// TIA Portal V17 export
// export: Created 2024-06-14T09:52:46.5071522Z, ExportSetting WithDefaults, DisplayName Totally Integrated Automation Portal, DisplayVersion V17, DisplayName TIA Portal Openness, DisplayVersion V17, DisplayName TIA Portal Version Control Interface, DisplayVersion V17, DisplayName Simotion SCOUT TIA, DisplayVersion 5.4.3.0, DisplayName SINAMICS Startdrive Advanced, DisplayVersion V17 SP1 Update 1, DisplayName SINAMICS Startdrive G110M, G120, G120C, G120D, G120P, G115D, DisplayVersion V17 SP1 Update 1, DisplayName SINAMICS Startdrive G130, G150, S120, S150, SINAMICS MV, S210, DisplayVersion V17 SP1 Update 1, DisplayName STEP 7 Professional, DisplayVersion V17, DisplayName STEP 7 Safety, DisplayVersion V17, DisplayName WinCC Professional, DisplayVersion V17
FUNCTION_BLOCK "Disable"   // FB3, LAD
{ S7_Optimized_Access := 'TRUE' }
VERSION : 0.1
// stored: AutoNumber false, IsIECCheckEnabled false, IsRetainMemResEnabled false, MemoryReserve 100, SetENOAutomatically false, UDAEnableTagReadback false
   VAR_INPUT
      Enable_Cylinder { ExternalAccessible := 'False'; ExternalVisible := 'False'; ExternalWritable := 'False'} : Array[1..6] of Bool;
      Enabled_Cylinder { ExternalAccessible := 'False'; ExternalVisible := 'False'; ExternalWritable := 'False'} : Int;
   END_VAR
   VAR_OUTPUT
      "First_Cylinder[1]" : Int;
      "First_Cylinder[2]" : Int;
      "First_Cylinder[3]" : Int;
      "First_Cylinder[4]" : Int;
      "First_Cylinder[5]" : Int;
      "First_Cylinder[6]" : Int;
      Disab_Total_Cyl : Int;
   END_VAR
   VAR
      Add_Cylinder : Array[1..6] of Int;
   END_VAR
   VAR_TEMP
      Temp8 : Int;
      Temp7 : Int;
      Temp6 : Int;
      Temp5 : Int;
      Temp4 : Int;
      Temp3 : Int;
      Temp2 : Int;
      Temp1 : Int;
      Temp9 : Int;
      Temp_8 : Int;
      Temp_7 : Int;
      Temp_6 : Int;
      Temp_5 : Int;
      Temp_4 : Int;
      Temp_3 : Int;
      Temp_2 : Int;
      Temp_1 : Int;
      Temp_9 : Int;
      Temp_91 : Int;
      Temp_81 : Int;
      Temp_71 : Int;
      Temp_61 : Int;
      Temp_51 : Int;
      Temp_41 : Int;
      Temp_31 : Int;
      Temp_21 : Int;
      Temp_11 : Int;
      Temp10 : Int;
      Temp_10 : Int;
      Temp_101 : Int;
   END_VAR
BEGIN

REGION Network 1: Disable Cylinder
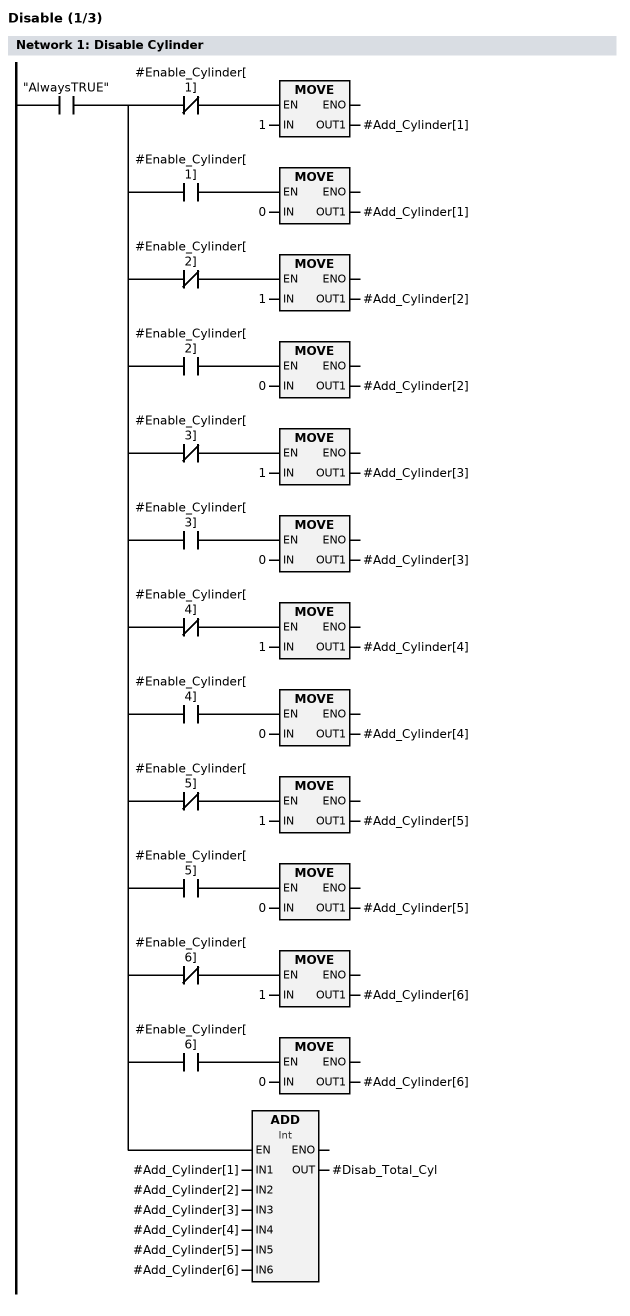
   RUNG wire#powerrail
      Contact( "AlwaysTRUE" )
      wire#w1
      I_Contact( #Enable_Cylinder[1] )
      Move(in := 1, out1 => #Add_Cylinder[1])
   END_RUNG
   RUNG wire#w1
      Contact( #Enable_Cylinder[1] )
      Move(in := 0, out1 => #Add_Cylinder[1])
   END_RUNG
   RUNG wire#w1
      I_Contact( #Enable_Cylinder[2] )
      Move(in := 1, out1 => #Add_Cylinder[2])
   END_RUNG
   RUNG wire#w1
      Contact( #Enable_Cylinder[2] )
      Move(in := 0, out1 => #Add_Cylinder[2])
   END_RUNG
   RUNG wire#w1
      I_Contact( #Enable_Cylinder[3] )
      Move(in := 1, out1 => #Add_Cylinder[3])
   END_RUNG
   RUNG wire#w1
      Contact( #Enable_Cylinder[3] )
      Move(in := 0, out1 => #Add_Cylinder[3])
   END_RUNG
   RUNG wire#w1
      I_Contact( #Enable_Cylinder[4] )
      Move(in := 1, out1 => #Add_Cylinder[4])
   END_RUNG
   RUNG wire#w1
      Contact( #Enable_Cylinder[4] )
      Move(in := 0, out1 => #Add_Cylinder[4])
   END_RUNG
   RUNG wire#w1
      I_Contact( #Enable_Cylinder[5] )
      Move(in := 1, out1 => #Add_Cylinder[5])
   END_RUNG
   RUNG wire#w1
      Contact( #Enable_Cylinder[5] )
      Move(in := 0, out1 => #Add_Cylinder[5])
   END_RUNG
   RUNG wire#w1
      I_Contact( #Enable_Cylinder[6] )
      Move(in := 1, out1 => #Add_Cylinder[6])
   END_RUNG
   RUNG wire#w1
      Contact( #Enable_Cylinder[6] )
      Move(in := 0, out1 => #Add_Cylinder[6])
   END_RUNG
   RUNG wire#w1
      { S7_Templates := "SrcType := Int" } Add(in1 := #Add_Cylinder[1], in2 := #Add_Cylinder[2], in3 := #Add_Cylinder[3], in4 := #Add_Cylinder[4], in5 := #Add_Cylinder[5], in6 := #Add_Cylinder[6], out => #Disab_Total_Cyl)
   END_RUNG
   // the same network as SCL:
   IF "AlwaysTRUE" AND NOT #Enable_Cylinder[1] THEN #Add_Cylinder[1] := 1; END_IF;
   IF "AlwaysTRUE" AND #Enable_Cylinder[1] THEN #Add_Cylinder[1] := 0; END_IF;
   IF "AlwaysTRUE" AND NOT #Enable_Cylinder[2] THEN #Add_Cylinder[2] := 1; END_IF;
   IF "AlwaysTRUE" AND #Enable_Cylinder[2] THEN #Add_Cylinder[2] := 0; END_IF;
   IF "AlwaysTRUE" AND NOT #Enable_Cylinder[3] THEN #Add_Cylinder[3] := 1; END_IF;
   IF "AlwaysTRUE" AND #Enable_Cylinder[3] THEN #Add_Cylinder[3] := 0; END_IF;
   IF "AlwaysTRUE" AND NOT #Enable_Cylinder[4] THEN #Add_Cylinder[4] := 1; END_IF;
   IF "AlwaysTRUE" AND #Enable_Cylinder[4] THEN #Add_Cylinder[4] := 0; END_IF;
   IF "AlwaysTRUE" AND NOT #Enable_Cylinder[5] THEN #Add_Cylinder[5] := 1; END_IF;
   IF "AlwaysTRUE" AND #Enable_Cylinder[5] THEN #Add_Cylinder[5] := 0; END_IF;
   IF "AlwaysTRUE" AND NOT #Enable_Cylinder[6] THEN #Add_Cylinder[6] := 1; END_IF;
   IF "AlwaysTRUE" AND #Enable_Cylinder[6] THEN #Add_Cylinder[6] := 0; END_IF;
   IF "AlwaysTRUE" THEN
       #Disab_Total_Cyl := #Add_Cylinder[1] + #Add_Cylinder[2] + #Add_Cylinder[3] + #Add_Cylinder[4] + #Add_Cylinder[5] + #Add_Cylinder[6];
   END_IF;
END_REGION

REGION Network 2: First Cylinder No-1
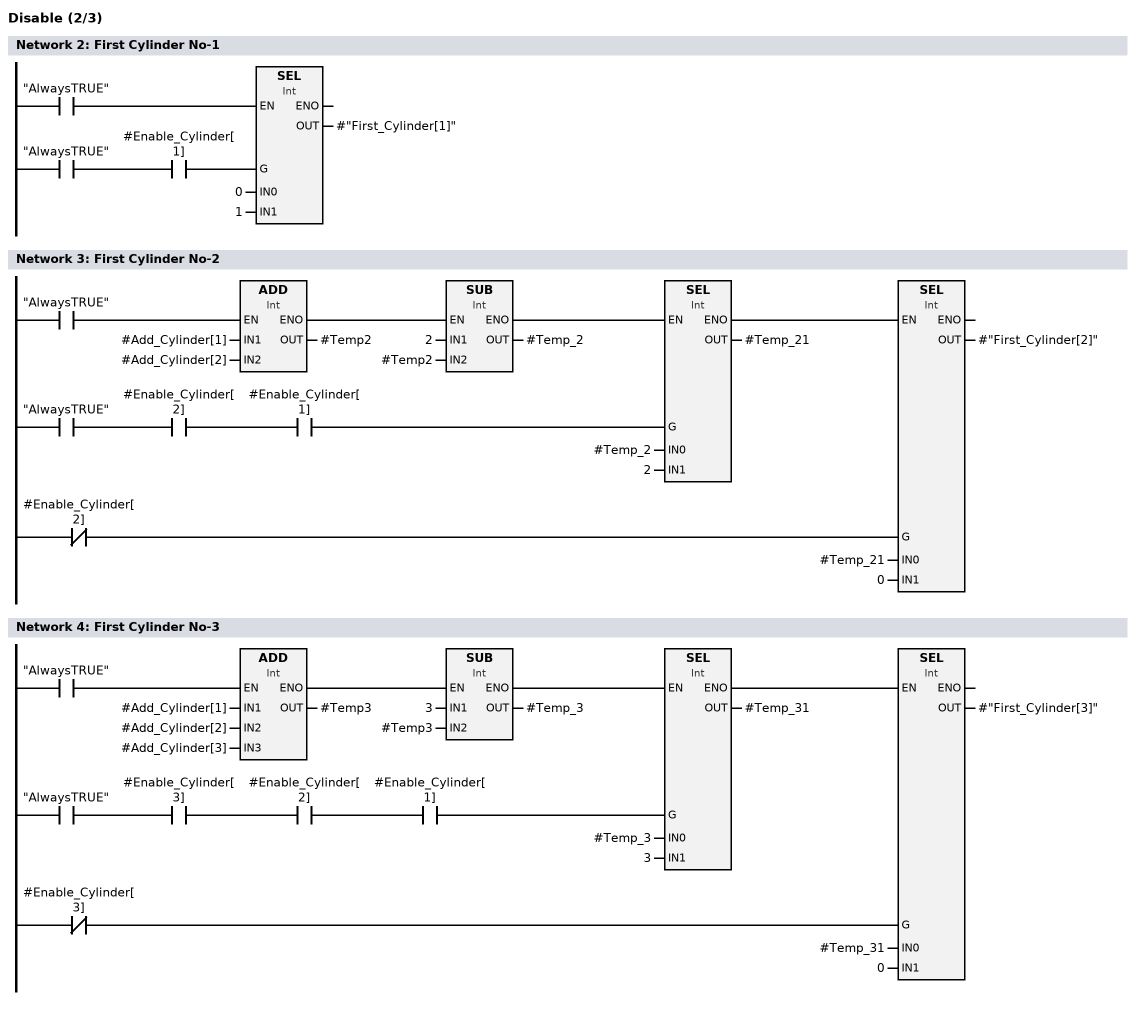
   RUNG wire#powerrail
      Contact( "AlwaysTRUE" )
      { S7_Templates := "value_type := Int" } SEL(g := wire#w1, in0 := 0, in1 := 1, out => #"First_Cylinder[1]")
   END_RUNG
   RUNG wire#powerrail
      Contact( "AlwaysTRUE" )
      Contact( #Enable_Cylinder[1] )
   END_RUNG wire#w1
   // the same network as SCL:
   IF "AlwaysTRUE" THEN
       #"First_Cylinder[1]" := SEL(G := "AlwaysTRUE" AND #Enable_Cylinder[1], IN0 := 0, IN1 := 1);
   END_IF;
END_REGION

REGION Network 3: First Cylinder No-2
   RUNG wire#powerrail
      Contact( "AlwaysTRUE" )
      { S7_Templates := "SrcType := Int" } Add(in1 := #Add_Cylinder[1], in2 := #Add_Cylinder[2], out => #Temp2)
      { S7_Templates := "SrcType := Int" } Sub(in1 := 2, in2 := #Temp2, out => #Temp_2)
      { S7_Templates := "value_type := Int" } SEL(g := wire#w1, in0 := #Temp_2, in1 := 2, out => #Temp_21)
      { S7_Templates := "value_type := Int" } SEL(g := wire#w2, in0 := #Temp_21, in1 := 0, out => #"First_Cylinder[2]")
   END_RUNG
   RUNG wire#powerrail
      Contact( "AlwaysTRUE" )
      Contact( #Enable_Cylinder[2] )
      Contact( #Enable_Cylinder[1] )
   END_RUNG wire#w1
   RUNG wire#powerrail
      I_Contact( #Enable_Cylinder[2] )
   END_RUNG wire#w2
   // the same network as SCL:
   // ENO of a box is taken as its EN; it also drops when the box reports an error
   IF "AlwaysTRUE" THEN
       #Temp2 := #Add_Cylinder[1] + #Add_Cylinder[2];
       #Temp_2 := 2 - #Temp2;
       #Temp_21 := SEL(G := "AlwaysTRUE" AND #Enable_Cylinder[2] AND #Enable_Cylinder[1], IN0 := #Temp_2, IN1 := 2);
       #"First_Cylinder[2]" := SEL(G := NOT #Enable_Cylinder[2], IN0 := #Temp_21, IN1 := 0);
   END_IF;
END_REGION

REGION Network 4: First Cylinder No-3
   RUNG wire#powerrail
      Contact( "AlwaysTRUE" )
      { S7_Templates := "SrcType := Int" } Add(in1 := #Add_Cylinder[1], in2 := #Add_Cylinder[2], in3 := #Add_Cylinder[3], out => #Temp3)
      { S7_Templates := "SrcType := Int" } Sub(in1 := 3, in2 := #Temp3, out => #Temp_3)
      { S7_Templates := "value_type := Int" } SEL(g := wire#w1, in0 := #Temp_3, in1 := 3, out => #Temp_31)
      { S7_Templates := "value_type := Int" } SEL(g := wire#w2, in0 := #Temp_31, in1 := 0, out => #"First_Cylinder[3]")
   END_RUNG
   RUNG wire#powerrail
      Contact( "AlwaysTRUE" )
      Contact( #Enable_Cylinder[3] )
      Contact( #Enable_Cylinder[2] )
      Contact( #Enable_Cylinder[1] )
   END_RUNG wire#w1
   RUNG wire#powerrail
      I_Contact( #Enable_Cylinder[3] )
   END_RUNG wire#w2
   // the same network as SCL:
   // ENO of a box is taken as its EN; it also drops when the box reports an error
   IF "AlwaysTRUE" THEN
       #Temp3 := #Add_Cylinder[1] + #Add_Cylinder[2] + #Add_Cylinder[3];
       #Temp_3 := 3 - #Temp3;
       #Temp_31 := SEL(G := "AlwaysTRUE" AND #Enable_Cylinder[3] AND #Enable_Cylinder[2] AND #Enable_Cylinder[1], IN0 := #Temp_3, IN1 := 3);
       #"First_Cylinder[3]" := SEL(G := NOT #Enable_Cylinder[3], IN0 := #Temp_31, IN1 := 0);
   END_IF;
END_REGION

REGION Network 5: First Cylinder No-4
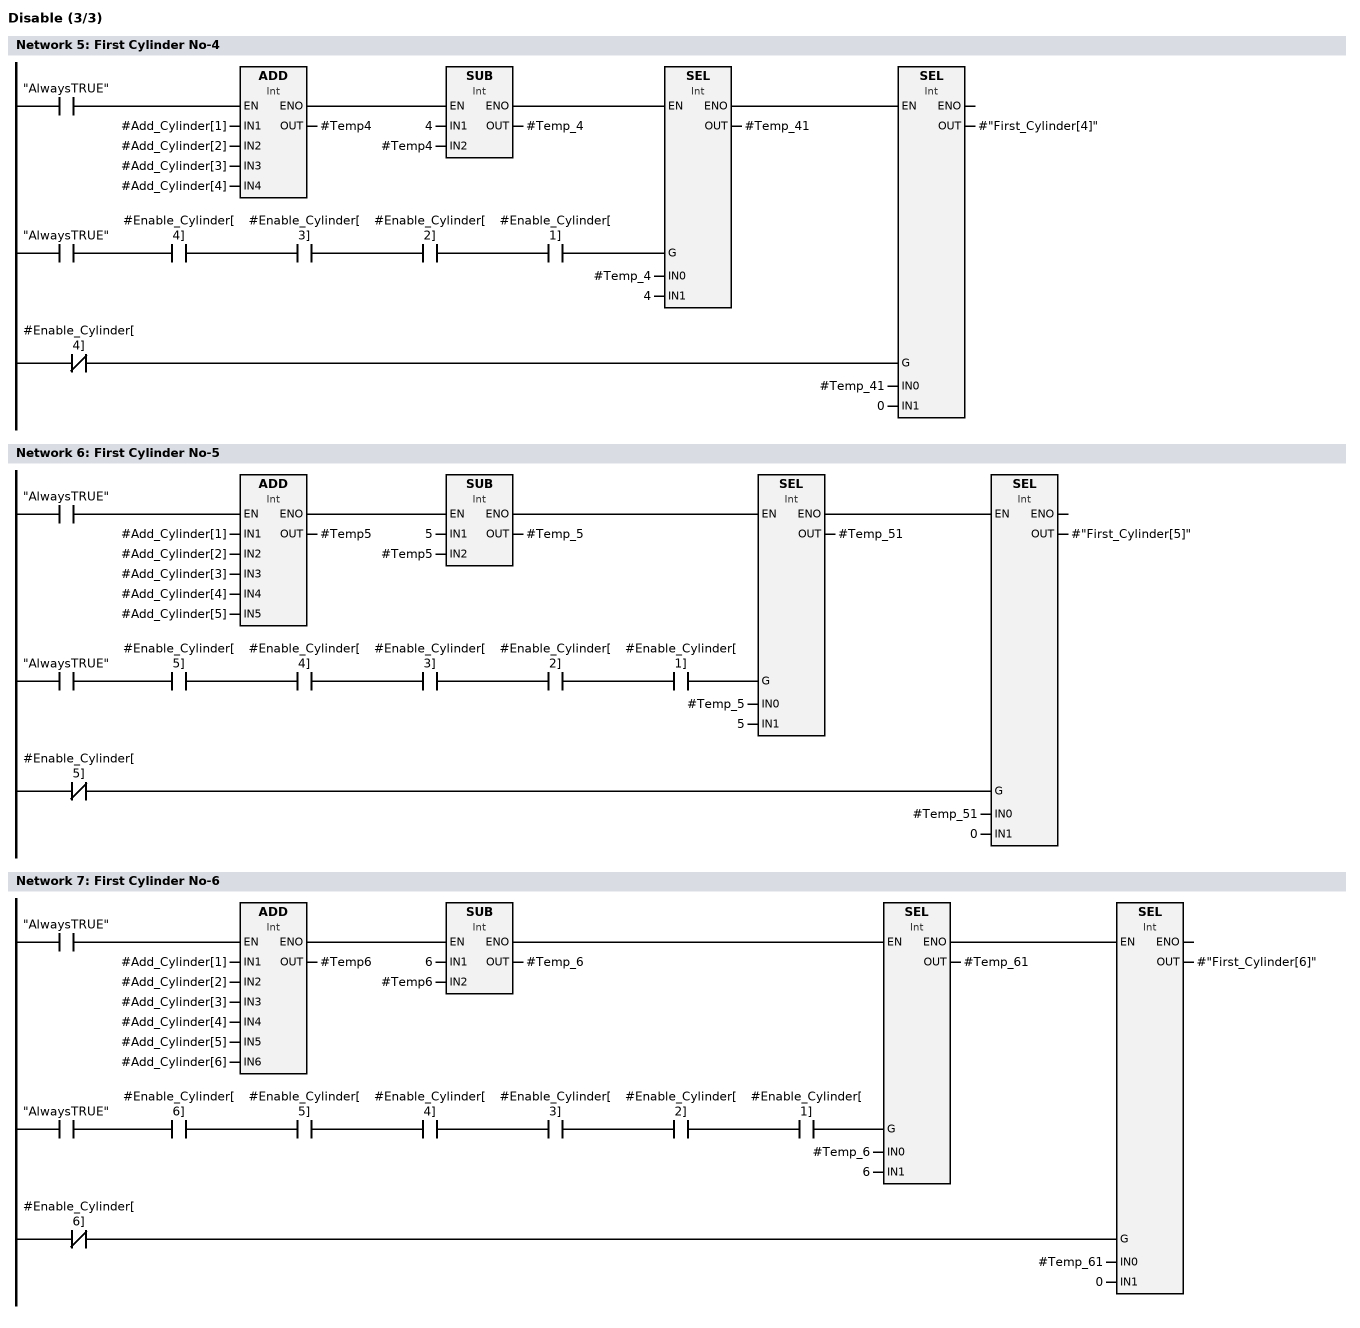
   RUNG wire#powerrail
      Contact( "AlwaysTRUE" )
      { S7_Templates := "SrcType := Int" } Add(in1 := #Add_Cylinder[1], in2 := #Add_Cylinder[2], in3 := #Add_Cylinder[3], in4 := #Add_Cylinder[4], out => #Temp4)
      { S7_Templates := "SrcType := Int" } Sub(in1 := 4, in2 := #Temp4, out => #Temp_4)
      { S7_Templates := "value_type := Int" } SEL(g := wire#w1, in0 := #Temp_4, in1 := 4, out => #Temp_41)
      { S7_Templates := "value_type := Int" } SEL(g := wire#w2, in0 := #Temp_41, in1 := 0, out => #"First_Cylinder[4]")
   END_RUNG
   RUNG wire#powerrail
      Contact( "AlwaysTRUE" )
      Contact( #Enable_Cylinder[4] )
      Contact( #Enable_Cylinder[3] )
      Contact( #Enable_Cylinder[2] )
      Contact( #Enable_Cylinder[1] )
   END_RUNG wire#w1
   RUNG wire#powerrail
      I_Contact( #Enable_Cylinder[4] )
   END_RUNG wire#w2
   // the same network as SCL:
   // ENO of a box is taken as its EN; it also drops when the box reports an error
   IF "AlwaysTRUE" THEN
       #Temp4 := #Add_Cylinder[1] + #Add_Cylinder[2] + #Add_Cylinder[3] + #Add_Cylinder[4];
       #Temp_4 := 4 - #Temp4;
       #Temp_41 := SEL(G := "AlwaysTRUE" AND #Enable_Cylinder[4] AND #Enable_Cylinder[3] AND #Enable_Cylinder[2] AND #Enable_Cylinder[1], IN0 := #Temp_4, IN1 := 4);
       #"First_Cylinder[4]" := SEL(G := NOT #Enable_Cylinder[4], IN0 := #Temp_41, IN1 := 0);
   END_IF;
END_REGION

REGION Network 6: First Cylinder No-5
   RUNG wire#powerrail
      Contact( "AlwaysTRUE" )
      { S7_Templates := "SrcType := Int" } Add(in1 := #Add_Cylinder[1], in2 := #Add_Cylinder[2], in3 := #Add_Cylinder[3], in4 := #Add_Cylinder[4], in5 := #Add_Cylinder[5], out => #Temp5)
      { S7_Templates := "SrcType := Int" } Sub(in1 := 5, in2 := #Temp5, out => #Temp_5)
      { S7_Templates := "value_type := Int" } SEL(g := wire#w1, in0 := #Temp_5, in1 := 5, out => #Temp_51)
      { S7_Templates := "value_type := Int" } SEL(g := wire#w2, in0 := #Temp_51, in1 := 0, out => #"First_Cylinder[5]")
   END_RUNG
   RUNG wire#powerrail
      Contact( "AlwaysTRUE" )
      Contact( #Enable_Cylinder[5] )
      Contact( #Enable_Cylinder[4] )
      Contact( #Enable_Cylinder[3] )
      Contact( #Enable_Cylinder[2] )
      Contact( #Enable_Cylinder[1] )
   END_RUNG wire#w1
   RUNG wire#powerrail
      I_Contact( #Enable_Cylinder[5] )
   END_RUNG wire#w2
   // the same network as SCL:
   // ENO of a box is taken as its EN; it also drops when the box reports an error
   IF "AlwaysTRUE" THEN
       #Temp5 := #Add_Cylinder[1] + #Add_Cylinder[2] + #Add_Cylinder[3] + #Add_Cylinder[4] + #Add_Cylinder[5];
       #Temp_5 := 5 - #Temp5;
       #Temp_51 := SEL(G := "AlwaysTRUE" AND #Enable_Cylinder[5] AND #Enable_Cylinder[4] AND #Enable_Cylinder[3] AND #Enable_Cylinder[2] AND #Enable_Cylinder[1], IN0 := #Temp_5, IN1 := 5);
       #"First_Cylinder[5]" := SEL(G := NOT #Enable_Cylinder[5], IN0 := #Temp_51, IN1 := 0);
   END_IF;
END_REGION

REGION Network 7: First Cylinder No-6
   RUNG wire#powerrail
      Contact( "AlwaysTRUE" )
      { S7_Templates := "SrcType := Int" } Add(in1 := #Add_Cylinder[1], in2 := #Add_Cylinder[2], in3 := #Add_Cylinder[3], in4 := #Add_Cylinder[4], in5 := #Add_Cylinder[5], in6 := #Add_Cylinder[6], out => #Temp6)
      { S7_Templates := "SrcType := Int" } Sub(in1 := 6, in2 := #Temp6, out => #Temp_6)
      { S7_Templates := "value_type := Int" } SEL(g := wire#w1, in0 := #Temp_6, in1 := 6, out => #Temp_61)
      { S7_Templates := "value_type := Int" } SEL(g := wire#w2, in0 := #Temp_61, in1 := 0, out => #"First_Cylinder[6]")
   END_RUNG
   RUNG wire#powerrail
      Contact( "AlwaysTRUE" )
      Contact( #Enable_Cylinder[6] )
      Contact( #Enable_Cylinder[5] )
      Contact( #Enable_Cylinder[4] )
      Contact( #Enable_Cylinder[3] )
      Contact( #Enable_Cylinder[2] )
      Contact( #Enable_Cylinder[1] )
   END_RUNG wire#w1
   RUNG wire#powerrail
      I_Contact( #Enable_Cylinder[6] )
   END_RUNG wire#w2
   // the same network as SCL:
   // ENO of a box is taken as its EN; it also drops when the box reports an error
   IF "AlwaysTRUE" THEN
       #Temp6 := #Add_Cylinder[1] + #Add_Cylinder[2] + #Add_Cylinder[3] + #Add_Cylinder[4] + #Add_Cylinder[5] + #Add_Cylinder[6];
       #Temp_6 := 6 - #Temp6;
       #Temp_61 := SEL(G := "AlwaysTRUE" AND #Enable_Cylinder[6] AND #Enable_Cylinder[5] AND #Enable_Cylinder[4] AND #Enable_Cylinder[3] AND #Enable_Cylinder[2] AND #Enable_Cylinder[1], IN0 := #Temp_6, IN1 := 6);
       #"First_Cylinder[6]" := SEL(G := NOT #Enable_Cylinder[6], IN0 := #Temp_61, IN1 := 0);
   END_IF;
END_REGION
END_FUNCTION_BLOCK
